RoboDK station: Deburring1.rdk

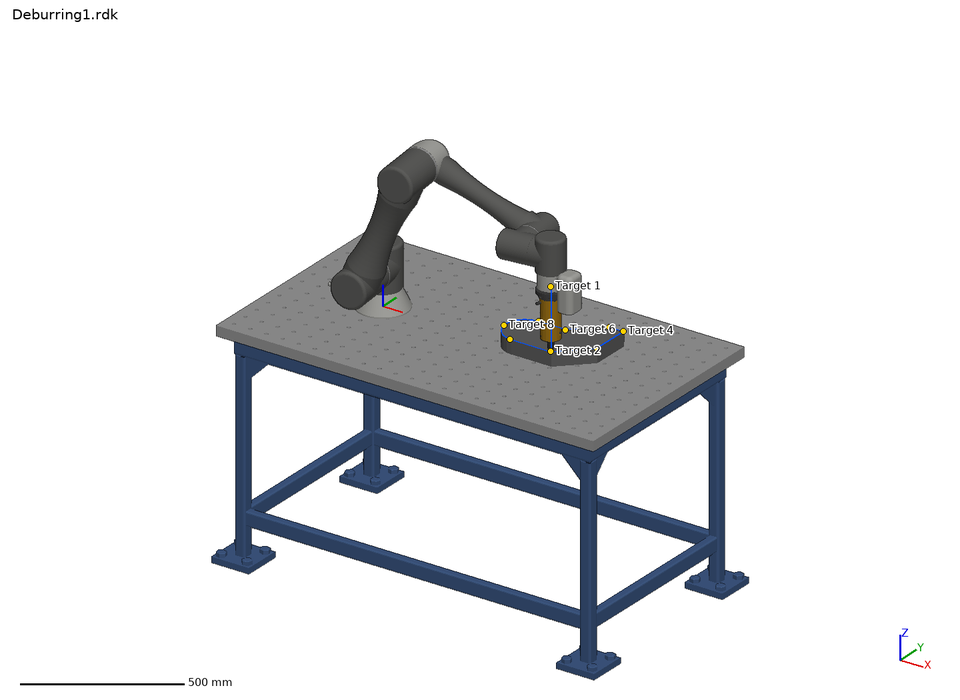
[picture v0: the station drawn from its stored meshes, robots at their saved joint values, targets as dots, program paths as lines]
Station Edge (saved by RoboDK 5.9.2). Poses are relative to the parent item; angles as X-Y-Z fixed-axis rotations.
  - frame TM5-900 Base at (0, 0, 0) mm
    - robot TM5-900: 6 axes, payload 4 kg, reach 900 mm, repeatability 0.1 mm, weight 30 kg
        modified DH rows (alpha deg, a mm, theta deg, d mm): 0, 0, 0, 145.2; 90, 0, 90, 0; 0, 429, 0, 0; 0, 411, -90, 122.3; -90, 0, 0, 106.5; 90, 0, 180, 114.15
        joint limits [-360, -180, -155, -180, -180, -270] to [360, 180, 155, 180, 180, 270]; home [0, 0, 90, -90, 90, 0]; saved at [6.131, 22.5, 90.557, -23.166, 89.988, 6.131]
      - tool ATI 9150-CDB-8-11-000 Deburring Tool (Spring), TCP at (0, 0, 215) mm, size 93.7 x 93.7 x 214.4 mm
    - target Target 1 (Cartesian target) at (658.82, -52.3, 271.64) mm, rotated rx 179.89 ry 0 rz 90 deg; joints [6.131, 18.221, 65.088, 6.582, 89.988, 6.131] of TM5-900
    - target Target 2 (Cartesian target) at (658.82, -52.3, 51.64) mm, rotated rx 179.89 ry 0 rz 90 deg; joints [6.131, 22.5, 90.557, -23.166, 89.988, 6.131] of TM5-900
    - target Target 3 (Cartesian target) at (758.82, 47.7, 51.64) mm, rotated rx 179.89 ry 0 rz 90 deg; joints [12.864, 35.398, 70.751, -16.256, 89.976, 12.864] of TM5-900
    - target Target 4 (Cartesian target) at (758.82, 187.7, 51.64) mm, rotated rx 179.89 ry 0 rz 90 deg; joints [22.913, 38.404, 65.792, -14.297, 89.957, 22.913] of TM5-900
    - target Target 5 (Cartesian target) at (708.82, 187.7, 51.64) mm, rotated rx 179.89 ry 0 rz 90 deg; joints [24.454, 31.752, 76.598, -18.45, 89.954, 24.454] of TM5-900
    - target Target 6 (Cartesian target) at (608.82, 97.7, 51.64) mm, rotated rx 179.89 ry 0 rz 90 deg; joints [20.578, 16.981, 98.204, -25.288, 89.961, 20.578] of TM5-900
    - target Target 7 (Cartesian target) at (508.82, 97.7, 51.64) mm, rotated rx 179.89 ry 0 rz 90 deg; joints [24.552, 4.426, 113.474, -28, 89.954, 24.552] of TM5-900
    - target Target 8 (Cartesian target) at (437.82, 17.7, 51.64) mm, rotated rx 179.89 ry 0 rz 90 deg; joints [18.55, -6.762, 124.395, -27.737, 89.965, 18.549] of TM5-900
    - target Target 9 (Cartesian target) at (507.82, -52.3, 51.64) mm, rotated rx 179.89 ry 0 rz 90 deg; joints [7.991, 3.414, 114.57, -28.093, 89.985, 7.991] of TM5-900
  - object Table 1400x800x800mm at (0, 0, 0) mm, size 1420 x 820 x 800 mm, geometry from Table-1400x800x800mm.sld
  - object random1 at (510, -50, 0) mm, size 325 x 240 x 50 mm, geometry from random1.step
  - program Prog1 (12 instructions, listed below)
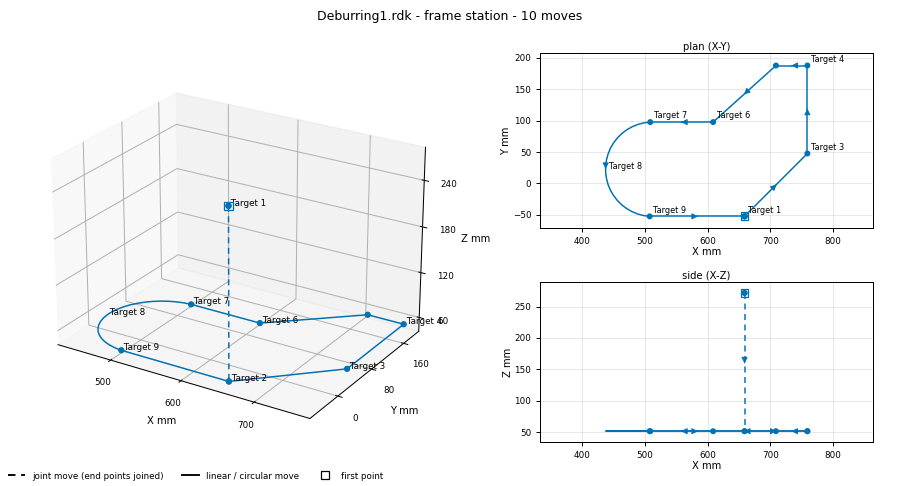
[picture p0: tool path of Deburring1.rdk in frame station, 10 of 10 moves have a stored position in this frame; points joined in program order, loops and branches not executed]

--- program Prog1 (robot TM5-900) ---
  Set Ref.: TM5-900 Base
  Set Tool: ATI 9150-CDB-8-11-000 Deburring Tool (Spring)
  MoveJ (Target 1)
  MoveJ (Target 1)
  MoveJ (Target 2)
  MoveL (Target 3)
  MoveL (Target 4)
  MoveL (Target 5)
  MoveL (Target 6)
  MoveL (Target 7)
  MoveC (Target 8, Target 9)
  MoveL (Target 2)
